TYPE Mechanical :
STRUCT
	rInputRev			:		REAL;
	rOutputRev			:		REAL;
	rScrewLead			:		REAL;
	rStroke				:		REAL;
END_STRUCT
END_TYPE

(* stored: Version 1.1.0.1, ProductVersion 3.1.4024.6
   DUT Mechanical: Id {54bd22e5-eafb-48ec-8949-13bf72bb4da7} *)
